// Struckig
// Copyright (C) 2022 Stefan Besler

// This program is free software: you can redistribute it and/or modify
// it under the terms of the GNU General Public License as published by
// the Free Software Foundation, either version 3 of the License, or
// (at your option) any later version.

// This program is distributed in the hope that it will be useful,
// but WITHOUT ANY WARRANTY; without even the implied warranty of
// MERCHANTABILITY or FITNESS FOR A PARTICULAR PURPOSE.  See the
// GNU General Public License for more details.
//
// You should have received a copy of the GNU General Public License
// along with THIS PROGRAM.  IF NOT, see <http://www.gnu.org/licenses/>.
/// Internal power helper that preserves sign for negative bases.
/// Evaluates `sign(v) * |v|^e`.
FUNCTION INTERNAL Power : LREAL
VAR_INPUT
  v : LREAL; //< Base value.
  e : LREAL; //< Exponent.
END_VAR

Power := SEL(v < 0, 1.0, -1.0) * EXPT(ABS(v), e);

END_FUNCTION

(* stored: Version 1.1.0.1
   POU Power: Id {76716193-d546-414d-a8ab-5cbcfa9a3d68}, SpecialFunc None *)
